TYPE ST_Position :
STRUCT
    nCol            : INT;
    nRow            : INT;
    fTargetX        : LREAL;
    fTargetY        : LREAL;
    bIsAisleStation : BOOL;
END_STRUCT
END_TYPE

(* stored: Version 1.1.0.1, ProductVersion 3.1.4024.16
   DUT ST_Position: Id {c9d0e1f2-a3b4-5678-2345-901234567890} *)
